// TIA Portal V20 export
TYPE "LKinCtrl_typePointParameter"
   STRUCT
      pathDynamics : "LKinCtrl_typePathDynamics";   // path dynamics for this command
      orientationDynamics : "LKinCtrl_typePathDynamics";   // orientation dynamics for this command
      orientationDirection : DInt := 3;   // 1: positive direction; 2: negative direction; 3: shortest distance
      bufferMode : DInt := 1;   // 1: standstill between commands, 2: blending with lower speed; 5: blending with higher speed
      transitionParameters : Array[1..5] of LReal;   // blending distance parameters
      dynamicAdaption : DInt := -1;   // <0.0: default TO setting used; 0: no dynamic adaption; 1: with variable limits; 2: with constant limits
      toolNumber : DInt;   // Tool number for SetTool command (LKINCTRL_MC_SETTOOL)
      moveDirectParameters : "LKinCtrl_typeMoveDirectParameter";   // parameters for MoveDirect command definition
      offsetParameters : "LKinCtrl_typeToolParameters";   // parameters for offset selection and configuration
      conveyorParameters : "LKinCtrl_typeConveyorParameter";   // parameters for conveyor selection and configuration
      circleParameters : "LKinCtrl_typeCircleParameters";   // parameters for circle command definition
      zoneParameters : "LKinCtrl_typeZoneParameters";   // parameters for zone commands
      pickAndPlaceParameters : "LKinCtrl_typeMovePickAndPlaceParameters";   // parameters for pick and place command
   END_STRUCT;
   // transitionParameters[1] := -1.0;
   // conveyorParameters.conveyorParaNo := 0;
END_TYPE
